ADAPTER HandshakeAdapter_Proposal (* Adapter Interface *)
  (* Standard: 61499-1 *)
  (* Version 0.0, 2/8/2021, prana, nxtControl GmbH *)
  PACKAGE Main;
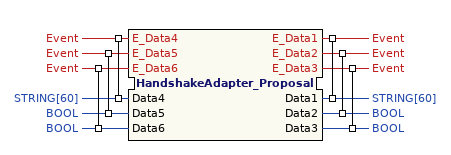
  EVENT_INPUT
    E_Data4 WITH Data4; (* Request from Socket *)
    E_Data5 WITH Data5;
    E_Data6 WITH Data6;
  END_EVENT
  EVENT_OUTPUT
    E_Data1 WITH Data1; (* Confirmation from Plug *)
    E_Data2 WITH Data2;
    E_Data3 WITH Data3;
  END_EVENT
  VAR_INPUT
    Data4 : STRING[60]; (* Request Data from Socket *)
    Data5 : BOOL;
    Data6 : BOOL;
  END_VAR
  VAR_OUTPUT
    Data1 : STRING[60]; (* Confirmation Data from Plug *)
    Data2 : BOOL;
    Data3 : BOOL;
  END_VAR
  SERVICE SOCKET/PLUG
    SEQUENCE request_confirm
      SOCKET.E_Data4(Data4) -> PLUG.E_Data4(Data4);
      PLUG.E_Data1(Data1) -> SOCKET.E_Data1(Data1);
    END_SEQUENCE
    SEQUENCE indication_response
      PLUG.IND(INDD) -> SOCKET.IND(INDD);
      SOCKET.RSP(RSPD) -> PLUG.RSP(RSPD);
    END_SEQUENCE
  END_SERVICE
END_ADAPTER
